// TwinCAT 3 PLC project TcoUtilities
// Title: TcoUtilities
// Company: Vortex.Library
// ProjectVersion: 0.6.0.913
// ProgramVersion: 3.1.4023.0
// libraries:
//   Tc2_Standard, * (Beckhoff Automation GmbH)
//   Tc2_System, * (Beckhoff Automation GmbH)
//   Tc3_Module, * (Beckhoff Automation GmbH)
//   TcoCore, 0.6.0.913 (Vortex.Library)
// project tree:
//   POUs/Conversions/ eTcoDataFormat.TcDUT
//   POUs/Conversions/FromBytes/ TcoBytesToDint.TcPOU, TcoBytesToUint.TcPOU, TcoBytesToUdint.TcPOU, TcoBytesToInt.TcPOU, TcoBytesToReal.TcPOU
//   POUs/Conversions/ToBytes/ TcoDintToBytes.TcPOU, TcoUintToBytes.TcPOU, TcoUdintToBytes.TcPOU, TcoIntToBytes.TcPOU, TcoRealToBytes.TcPOU
//   POUs/TcoEvaluvateMeasurement/ TcoEvaluateMeasurementDataItem.TcDUT, TcoEvaluateMeasurementTask.TcPOU, TcoEvaluateMeasurementResults.TcDUT, TcoEvaluateMeasurementConfig.TcDUT
//   POUs/TcoBlinker/ TcoBlinker.TcPOU
//   POUs/ TcoGetBitFromByte.TcPOU, TcoSetBitInByte.TcPOU
// real-time tasks:
//   TASK PlcTask: cycle T#10ms, priority 20, ADS port 350
//   TASK PlcTask1: cycle T#10ms, priority 21, ADS port 351

// ---- POUs/Conversions/eTcoDataFormat.TcDUT
{attribute 'qualified_only'}
{attribute 'strict'}
TYPE eTcoDataFormat :
(
    LittleEndian := 1,
    BigEndian := 2
);
END_TYPE

// ---- POUs/TcoEvaluvateMeasurement/TcoEvaluateMeasurementDataItem.TcDUT
TYPE TcoEvaluateMeasurementDataItem :
STRUCT
    TimeBase : TIME;
    Distance : REAL;
    ProcessValue : REAL;
    DiscreteValue : REAL;
END_STRUCT
END_TYPE

// ---- POUs/TcoEvaluvateMeasurement/TcoEvaluateMeasurementResults.TcDUT
TYPE TcoEvaluateMeasurementResults :
STRUCT
    RisingPeaks : ARRAY[0..100] OF TcoEvaluateMeasurementDataItem;
    RisingPeaksFound : INT;
    FallingPeaks : ARRAY[0..100] OF TcoEvaluateMeasurementDataItem;
    FallingPeaksFound : INT;
    Triggers : ARRAY[0..100] OF TcoEvaluateMeasurementDataItem;
    TriggersFound : INT;
END_STRUCT
END_TYPE

// ---- POUs/TcoEvaluvateMeasurement/TcoEvaluateMeasurementConfig.TcDUT
{attribute wpf [Container(Layout.Stack)]}
{attribute wpf [Group(Layout.GroupBox)]}
TYPE TcoEvaluateMeasurementConfig :
STRUCT
    {attribute wpf [Container(Layout.Stack, "FILTER")]}
    FilterValue : INT;
    {attribute wpf [Container(Layout.Stack, "SEARCH RANGE")]}
    SearchRange : INT;
    {attribute wpf [Container(Layout.Stack, "PEAK NOISE")]}
    PeaksNoise : REAL;
    {attribute wpf [Container(Layout.Stack, "TRIGGER NOISE")]}
    TriggerNoise : REAL;
    {attribute wpf [Container(Layout.Stack, "SMOOT FACTOR")]}
    SmoothFactor : REAL;
    {attribute wpf [Container(Layout.Stack, "NUMBER OF SAMPLES TO IGNORE - START")]}
    IgnoreSamplesFromStart : INT;
    {attribute wpf [Container(Layout.Stack, "NUMBER OF SAMPLES TO IGNORE - END")]}
    IgnoreSamplesFromEnd : INT;
    {attribute wpf [Container(Layout.Stack, "IGNORE ZERO VALUES - TIME BASE")]}
    IgnoreZeroSamplesIfTimeBase : BOOL;
    {attribute wpf [Container(Layout.Stack, "IGNORE ZERO VALUES - DISTANCE")]}
    IgnoreZeroSamplesIfDistance : BOOL;
    {attribute wpf [Container(Layout.Stack, "MAX FOUND LIMIT EXTREMS (MAX 100)(PROCES DATA ROW)")]}
    LimitIndexFoundExtrems : INT;
    {attribute wpf [Container(Layout.Stack, "MAX FOUND LIMIT TRIGGERS (MAX 100) (DISCRETE DATA ROW)")]}
    LimitIndexFoundTriggers : INT;
    {attribute wpf [Container(Layout.Stack, "PROCESS VALUE ROW NAME")]}
    ProcessValueRowName : STRING;
    {attribute wpf [Container(Layout.Stack, "DISCRETE VALUE ROW NAME")]}
    DiscreteValueRowName : STRING;
    {attribute wpf [Container(Layout.Stack, "EXPORT RAW DATA LOCATION")]}
    ExportRawLocation : STRING(255);
    {attribute wpf [Container(Layout.Stack, "EXPORT RESULTS LOCATION")]}
    ExportResultsLocation : STRING(255);
END_STRUCT
END_TYPE

// ---- POUs/Conversions/FromBytes/TcoBytesToDint.TcPOU
FUNCTION TcoBytesToDint : DINT
VAR_INPUT
    inFormat : eTcoDataFormat;
    inByte0 : BYTE;
    inByte1 : BYTE;
    inByte2 : BYTE;
    inByte3 : BYTE;
END_VAR
VAR
    _b0 : BYTE;
    _b1 : BYTE;
    _b2 : BYTE;
    _b3 : BYTE;
    _tmpDWORD : DWORD;
END_VAR

IF inFormat = eTcoDataFormat.LittleEndian THEN
    _b0 := inByte3;
    _b1 := inByte2;
    _b2 := inByte1;
    _b3 := inByte0;
ELSIF inFormat = eTcoDataFormat.BigEndian THEN
    _b0 := inByte0;
    _b1 := inByte1;
    _b2 := inByte2;
    _b3 := inByte3;
END_IF

_tmpDWORD := _b0;
_tmpDWORD := SHL(_tmpDWORD, 8);
_tmpDWORD := _tmpDWORD + _b1;
_tmpDWORD := SHL(_tmpDWORD, 8);
_tmpDWORD := _tmpDWORD + _b2;
_tmpDWORD := SHL(_tmpDWORD, 8);
_tmpDWORD := _tmpDWORD + _b3;
TcoBytesToDint := DWORD_TO_DINT(_tmpDWORD);

END_FUNCTION

// ---- POUs/Conversions/FromBytes/TcoBytesToUint.TcPOU
FUNCTION TcoBytesToUint : UINT
VAR_INPUT
    inFormat : eTcoDataFormat;
    inByte0 : BYTE;
    inByte1 : BYTE;
END_VAR
VAR
    _b0 : BYTE;
    _b1 : BYTE;
    _tmpWORD : WORD;
END_VAR

IF inFormat = eTcoDataFormat.LittleEndian THEN
    _b0 := inByte1;
    _b1 := inByte0;
ELSIF inFormat = eTcoDataFormat.BigEndian THEN
    _b0 := inByte0;
    _b1 := inByte1;
END_IF

_tmpWORD := _b0;
_tmpWORD := SHL(_tmpWORD, 8);
_tmpWORD := _tmpWORD + _b1;
TcoBytesToUint := WORD_TO_UINT(_tmpWORD);

END_FUNCTION

// ---- POUs/Conversions/FromBytes/TcoBytesToUdint.TcPOU
FUNCTION TcoBytesToUdint : UDINT
VAR_INPUT
    inFormat : eTcoDataFormat;
    inByte0 : BYTE;
    inByte1 : BYTE;
    inByte2 : BYTE;
    inByte3 : BYTE;
END_VAR
VAR
    _b0 : BYTE;
    _b1 : BYTE;
    _b2 : BYTE;
    _b3 : BYTE;
    _tmpDWORD : DWORD;
END_VAR

IF inFormat = eTcoDataFormat.LittleEndian THEN
    _b0 := inByte3;
    _b1 := inByte2;
    _b2 := inByte1;
    _b3 := inByte0;
ELSIF inFormat = eTcoDataFormat.BigEndian THEN
    _b0 := inByte0;
    _b1 := inByte1;
    _b2 := inByte2;
    _b3 := inByte3;
END_IF

_tmpDWORD := _b0;
_tmpDWORD := SHL(_tmpDWORD, 8);
_tmpDWORD := _tmpDWORD + _b1;
_tmpDWORD := SHL(_tmpDWORD, 8);
_tmpDWORD := _tmpDWORD + _b2;
_tmpDWORD := SHL(_tmpDWORD, 8);
_tmpDWORD := _tmpDWORD + _b3;
TcoBytesToUdint := DWORD_TO_UDINT(_tmpDWORD);

END_FUNCTION

// ---- POUs/Conversions/FromBytes/TcoBytesToInt.TcPOU
FUNCTION TcoBytesToInt : INT
VAR_INPUT
    inFormat : eTcoDataFormat;
    inByte0 : BYTE;
    inByte1 : BYTE;
END_VAR
VAR
    _b0 : BYTE;
    _b1 : BYTE;
    _tmpWORD : WORD;
END_VAR

IF inFormat = eTcoDataFormat.LittleEndian THEN
    _b0 := inByte1;
    _b1 := inByte0;
ELSIF inFormat = eTcoDataFormat.BigEndian THEN
    _b0 := inByte0;
    _b1 := inByte1;
END_IF

_tmpWORD := _b0;
_tmpWORD := SHL(_tmpWORD, 8);
_tmpWORD := _tmpWORD + _b1;
TcoBytesToInt := WORD_TO_INT(_tmpWORD);

END_FUNCTION

// ---- POUs/Conversions/FromBytes/TcoBytesToReal.TcPOU
FUNCTION TcoBytesToReal : REAL
VAR_INPUT
    inFormat : eTcoDataFormat;
    inByte0 : BYTE;
    inByte1 : BYTE;
    inByte2 : BYTE;
    inByte3 : BYTE;
END_VAR
VAR
    _b0 : BYTE;
    _b1 : BYTE;
    _b2 : BYTE;
    _b3 : BYTE;
    _w0 : WORD;
    _w1 : WORD;
    _Sign : DINT;
    _Exponent : DINT;
    _Fraction : REAL;
    _retval : LREAL;
END_VAR

IF inFormat = eTcoDataFormat.LittleEndian THEN
    _b0 := inByte3;
    _b1 := inByte2;
    _b2 := inByte1;
    _b3 := inByte0;
ELSIF inFormat = eTcoDataFormat.BigEndian THEN
    _b0 := inByte0;
    _b1 := inByte1;
    _b2 := inByte2;
    _b3 := inByte3;
END_IF

IF _b0 = 0 AND _b1 = 0 AND _b2 = 0 AND _b3 = 0 THEN
    TcoBytesToReal := 0;
    return;
END_IF

_w0 := 256 * _b0 + _b1;
_w1 := 256 * _b2 + _b3;
_Sign := SHR(_w0, 15);
_Exponent := SHR(SHL(_w0, 1), 8);
_Fraction := ANY_TO_REAL((SHR(SHL(_w0, 9), 9) * 65536) + _w1) / 8388608;
_retval := LREAL_TO_REAL(EXPT(-1, _Sign) * EXPT(2, _Exponent - 127) * (_Fraction + 1.0));

IF (_retval <= -EXPT(2, 128)) OR (_retval >= EXPT(2, 128)) THEN
    _retval := 0;
END_IF

TcoBytesToReal := _retval;

END_FUNCTION

// ---- POUs/Conversions/ToBytes/TcoDintToBytes.TcPOU
FUNCTION TcoDintToBytes
VAR_INPUT
    inFormat : eTcoDataFormat;
    inValue : DINT;
END_VAR
VAR_IN_OUT
    outByte0 : BYTE;
    outByte1 : BYTE;
    outByte2 : BYTE;
    outByte3 : BYTE;
END_VAR
VAR
    _b0 : BYTE;
    _b1 : BYTE;
    _b2 : BYTE;
    _b3 : BYTE;
    _tmpDINT : DINT;
END_VAR

_tmpDINT := inValue;
_b3 := UDINT_TO_BYTE(_tmpDINT MOD 256);
_tmpDINT := SHR(_tmpDINT, 8);
_b2 := UDINT_TO_BYTE(_tmpDINT MOD 256);
_tmpDINT := SHR(_tmpDINT, 8);
_b1 := UDINT_TO_BYTE(_tmpDINT MOD 256);
_tmpDINT := SHR(_tmpDINT, 8);
_b0 := UDINT_TO_BYTE(_tmpDINT MOD 256);
_tmpDINT := SHR(_tmpDINT, 8);

IF inFormat = eTcoDataFormat.LittleEndian THEN
    outByte0 := _b3;
    outByte1 := _b2;
    outByte2 := _b1;
    outByte3 := _b0;
ELSIF inFormat = eTcoDataFormat.BigEndian THEN
    outByte0 := _b0;
    outByte1 := _b1;
    outByte2 := _b2;
    outByte3 := _b3;
END_IF

END_FUNCTION

// ---- POUs/Conversions/ToBytes/TcoUintToBytes.TcPOU
FUNCTION TcoUintToBytes
VAR_INPUT
    inFormat : eTcoDataFormat;
    inValue : UINT;
END_VAR
VAR_IN_OUT
    outByte0 : BYTE;
    outByte1 : BYTE;
END_VAR
VAR
    _b0 : BYTE;
    _b1 : BYTE;
    _tmpUINT : UINT;
END_VAR

_tmpUINT := inValue;
_b1 := UDINT_TO_BYTE(_tmpUINT MOD 256);
_tmpUINT := SHR(_tmpUINT, 8);
_b0 := UDINT_TO_BYTE(_tmpUINT MOD 256);
_tmpUINT := SHR(_tmpUINT, 8);

IF inFormat = eTcoDataFormat.LittleEndian THEN
    outByte0 := _b1;
    outByte1 := _b0;
ELSIF inFormat = eTcoDataFormat.BigEndian THEN
    outByte0 := _b0;
    outByte1 := _b1;
END_IF

END_FUNCTION

// ---- POUs/Conversions/ToBytes/TcoUdintToBytes.TcPOU
FUNCTION TcoUdintToBytes
VAR_INPUT
    inFormat : eTcoDataFormat;
    inValue : UDINT;
END_VAR
VAR_IN_OUT
    outByte0 : BYTE;
    outByte1 : BYTE;
    outByte2 : BYTE;
    outByte3 : BYTE;
END_VAR
VAR
    _b0 : BYTE;
    _b1 : BYTE;
    _b2 : BYTE;
    _b3 : BYTE;
    _tmpUDINT : UDINT;
END_VAR

_tmpUDINT := inValue;
_b3 := UDINT_TO_BYTE(_tmpUDINT MOD 256);
_tmpUDINT := SHR(_tmpUDINT, 8);
_b2 := UDINT_TO_BYTE(_tmpUDINT MOD 256);
_tmpUDINT := SHR(_tmpUDINT, 8);
_b1 := UDINT_TO_BYTE(_tmpUDINT MOD 256);
_tmpUDINT := SHR(_tmpUDINT, 8);
_b0 := UDINT_TO_BYTE(_tmpUDINT MOD 256);
_tmpUDINT := SHR(_tmpUDINT, 8);

IF inFormat = eTcoDataFormat.LittleEndian THEN
    outByte0 := _b3;
    outByte1 := _b2;
    outByte2 := _b1;
    outByte3 := _b0;
ELSIF inFormat = eTcoDataFormat.BigEndian THEN
    outByte0 := _b0;
    outByte1 := _b1;
    outByte2 := _b2;
    outByte3 := _b3;
END_IF

END_FUNCTION

// ---- POUs/Conversions/ToBytes/TcoIntToBytes.TcPOU
FUNCTION TcoIntToBytes
VAR_INPUT
    inFormat : eTcoDataFormat;
    inValue : INT;
END_VAR
VAR_IN_OUT
    outByte0 : BYTE;
    outByte1 : BYTE;
END_VAR
VAR
    _b0 : BYTE;
    _b1 : BYTE;
    _tmpINT : INT;
END_VAR

_tmpINT := inValue;
_b1 := UDINT_TO_BYTE(_tmpINT MOD 256);
_tmpINT := SHR(_tmpINT, 8);
_b0 := UDINT_TO_BYTE(_tmpINT MOD 256);
_tmpINT := SHR(_tmpINT, 8);

IF inFormat = eTcoDataFormat.LittleEndian THEN
    outByte0 := _b1;
    outByte1 := _b0;
ELSIF inFormat = eTcoDataFormat.BigEndian THEN
    outByte0 := _b0;
    outByte1 := _b1;
END_IF

END_FUNCTION

// ---- POUs/Conversions/ToBytes/TcoRealToBytes.TcPOU
FUNCTION TcoRealToBytes
VAR_INPUT
    inFormat : eTcoDataFormat;
    inValue : REAL;
END_VAR
VAR_IN_OUT
    outByte0 : BYTE;
    outByte1 : BYTE;
    outByte2 : BYTE;
    outByte3 : BYTE;
END_VAR
VAR
    _b0 : BYTE;
    _b1 : BYTE;
    _b2 : BYTE;
    _b3 : BYTE;
    _tmpReal : REAL;
    _rExponent : LREAL;
    _Exponent : DINT;
    _Fraction : DINT;
    _tmpDINT : DINT;
END_VAR

IF (inValue <= -EXPT(2, 128)) OR (inValue >= EXPT(2, 128)) THEN
    outByte0 := 0;
    outByte1 := 0;
    outByte2 := 0;
    outByte3 := 0;
    return;
END_IF

IF inValue < 0 THEN
    _tmpReal := ABS(inValue);
    _rExponent := LOG(_tmpReal) / LOG(2);

    IF _rExponent >= 0 THEN
        _Exponent := TRUNC(_rExponent);
    ELSE
        _Exponent := TRUNC(_rExponent) - 1;
    END_IF

    _Fraction := REAL_TO_DINT((_tmpReal / EXPT(2, _Exponent) - 1) * 8388608);
    _tmpDINT := ANY_TO_DINT(2147483648 + (_Exponent + 127) * 8388608 + _Fraction);
ELSIF inValue > 0 THEN
    _tmpReal := ABS(inValue);
    _rExponent := LOG(_tmpReal) / LOG(2);

    IF _rExponent >= 0 THEN
        _Exponent := TRUNC(_rExponent);
    ELSE
        _Exponent := TRUNC(_rExponent) - 1;
    END_IF

    _Fraction := REAL_TO_DINT((_tmpReal / EXPT(2, _Exponent) - 1) * 8388608);
    _tmpDINT := ANY_TO_DINT((_Exponent + 127) * 8388608 + _Fraction);
ELSE
    _tmpDINT := 0;
END_IF

_b3 := UDINT_TO_BYTE(_tmpDINT MOD 256);
_tmpDINT := SHR(_tmpDINT, 8);
_b2 := UDINT_TO_BYTE(_tmpDINT MOD 256);
_tmpDINT := SHR(_tmpDINT, 8);
_b1 := UDINT_TO_BYTE(_tmpDINT MOD 256);
_tmpDINT := SHR(_tmpDINT, 8);
_b0 := UDINT_TO_BYTE(_tmpDINT MOD 256);
_tmpDINT := SHR(_tmpDINT, 8);

IF inFormat = eTcoDataFormat.LittleEndian THEN
    outByte0 := _b3;
    outByte1 := _b2;
    outByte2 := _b1;
    outByte3 := _b0;
ELSIF inFormat = eTcoDataFormat.BigEndian THEN
    outByte0 := _b0;
    outByte1 := _b1;
    outByte2 := _b2;
    outByte3 := _b3;
END_IF

END_FUNCTION

// ---- POUs/TcoEvaluvateMeasurement/TcoEvaluateMeasurementTask.TcPOU
FUNCTION_BLOCK TcoEvaluateMeasurementTask EXTENDS TcoCore.TcoRemoteTask
VAR
    _config : TcoEvaluateMeasurementConfig;
    _data : ARRAY[0..1000] OF TcoEvaluateMeasurementDataItem;
    _results : TcoEvaluateMeasurementResults;
    _entityId : STRING;
    {attribute 'hide'}
    _cleanResultData : TcoEvaluateMeasurementResults;
    {attribute 'hide'}
    _cleanData : ARRAY[0..1000] OF TcoEvaluateMeasurementDataItem;
END_VAR

SUPER^();

PROPERTY Config : TcoEvaluateMeasurementConfig
GET
Config := _config;
END_GET
END_PROPERTY

PROPERTY DataSource : ARRAY[0..1000] OF TcoEvaluateMeasurementDataItem
GET
DataSource := _data;
END_GET
SET
_data := DataSource;
END_SET
END_PROPERTY

(*~
    <docu>
        <summary>
            Restores this instance to the Ready state. Can be called explicitly or from within one of the restore mechanisms.
            <para>
                See also <see cref="PlcDocu.TcoCore.TcoTask.AutoRestorable()"/>
            </para>
        </summary>
    </docu>
~*)
METHOD Restore : ITcoRestorable
SUPER^.Restore();
_data := _cleanData;
_results := _cleanResultData;
END_METHOD

PROPERTY Results : TcoEvaluateMeasurementResults
GET
Results := _results;
END_GET
END_PROPERTY

METHOD Run : REFERENCE TO TcoEvaluateMeasurementTask
VAR_INPUT
    inEntityId : STRING;
    inConfig : TcoEvaluateMeasurementConfig;
    inData : ARRAY[0..1000] OF TcoEvaluateMeasurementDataItem;
END_VAR
VAR
    _cleanResultData : TcoEvaluateMeasurementResults;
END_VAR
_config := inConfig;
_entityId := inEntityId;
_data := inData;
Run REF= THIS^;
END_METHOD

END_FUNCTION_BLOCK

// ---- POUs/TcoBlinker/TcoBlinker.TcPOU
(*~
    <docu>
        <summary>
            Provides periodic on/off switcher.
        </summary>
    </docu>
~*)
FUNCTION_BLOCK TcoBlinker EXTENDS TcoCore.TcoObject
VAR_INPUT
    (*~
        <docu>
            <summary>
                Time duration for on duty output.
            </summary>
        </docu>
    ~*)
    inOnTime : TIME;
    (*~
        <docu>
            <summary>
                Time duration for off duty output.
            </summary>
        </docu>
    ~*)
    inOffTime : TIME;
END_VAR
VAR_OUTPUT
    outQ : BOOL;
END_VAR
VAR
    {attribute 'hide'}
    _onTimer : TON;
    {attribute 'hide'}
    _offTimer : TON;
    {attribute 'hide'}
    _nextExpectedCycle : ULINT;
    {attribute 'hide'}
    _state : INT;
END_VAR

IF (THIS^.Context.StartCycleCount <> _nextExpectedCycle) THEN
    _state := 0;
END_IF

_nextExpectedCycle := THIS^.Context.StartCycleCount + 1;

IF (_state = 0) THEN
    _offTimer(IN := FALSE);
    _onTimer(IN := FALSE);
    _state := 1;
END_IF;

IF (_state = 1) THEN
    _onTimer(IN := TRUE, PT := inOnTime);
    outQ := TRUE;

    IF (_onTimer.Q) THEN
        _state := 2;
        RETURN;
    END_IF;
END_IF;

IF (_state = 2) THEN
    _offTimer(IN := TRUE, PT := inOffTime);
    outQ := FALSE;

    IF (_offTimer.Q) THEN
        _state := 0;
    END_IF;
END_IF

{attribute 'hide'}
METHOD FB_init : BOOL
VAR_INPUT
    bInitRetains : BOOL; // if TRUE, the retain variables are initialized (warm start / cold start)
    bInCopyCode : BOOL; // if TRUE, the instance afterwards gets moved into the copy code (online change)
    ParentObject : ITcoObject;
END_VAR
END_METHOD

(*~
    <docu>
        <summary>
            Gets `true` when the switcher is in off duty phase.
        </summary>
    </docu>
~*)
PROPERTY IsOff : BOOL
GET
IsOff := NOT outQ;
END_GET
END_PROPERTY

(*~
    <docu>
        <summary>
            Gets `true` when the switcher is in on duty phase.
        </summary>
    </docu>
~*)
PROPERTY IsOn : BOOL
GET
IsOn := outQ;
END_GET
END_PROPERTY

END_FUNCTION_BLOCK

// ---- POUs/TcoGetBitFromByte.TcPOU
FUNCTION TcoGetBitFromByte : BOOL
VAR_INPUT
    inByteValue : BYTE;
    inBit : UINT;
END_VAR

TcoGetBitFromByte := FALSE;

CASE inBit OF
    0:
        TcoGetBitFromByte := inByteValue.0;
    1:
        TcoGetBitFromByte := inByteValue.1;
    2:
        TcoGetBitFromByte := inByteValue.2;
    3:
        TcoGetBitFromByte := inByteValue.3;
    4:
        TcoGetBitFromByte := inByteValue.4;
    5:
        TcoGetBitFromByte := inByteValue.5;
    6:
        TcoGetBitFromByte := inByteValue.6;
    7:
        TcoGetBitFromByte := inByteValue.7;
END_CASE

END_FUNCTION

// ---- POUs/TcoSetBitInByte.TcPOU
FUNCTION TcoSetBitInByte
VAR_INPUT
    inBitValue : BOOL;
    inBit : UINT;
END_VAR
VAR_IN_OUT
    inoOut : BYTE;
END_VAR

CASE inBit OF
    0:
        inoOut.0 := inBitValue;
    1:
        inoOut.1 := inBitValue;
    2:
        inoOut.2 := inBitValue;
    3:
        inoOut.3 := inBitValue;
    4:
        inoOut.4 := inBitValue;
    5:
        inoOut.5 := inBitValue;
    6:
        inoOut.6 := inBitValue;
    7:
        inoOut.7 := inBitValue;
END_CASE

END_FUNCTION
